	            "FC_Statistics"(ix_Reset := #iUDT_EquipmentControl.Command.ResetData,        // Reset statistics input
	                            ix_Activate := NOT #sx_safetyZoneOk,                                    // Activate statistics functions input
	                            ix_RTrigActivate := #sR_TRIG_NotHealthy.Q,                                   // Statistics active trigger
	                            iqUDT_Statistics := #iqUDT_Statistics.NotHealthy);                       // Statistics values output
	        END_IF;

	    END_REGION

	END_REGION



END_FUNCTION_BLOCK

FUNCTION_BLOCK "FB_UPSThreatParcel"
{ S7_Optimized_Access := 'TRUE' }
VERSION : 0.1
// ATTRIBUTES
// AUTO_NUMBER = True
// BLOCK_NUMBER = 63
// END_ATTRIBUTES
   VAR_INPUT
      ii_TrackingPosition { ExternalAccessible := 'False'; ExternalVisible := 'False'; ExternalWritable := 'False'} : Int;
      ix_ReleaseButton { ExternalAccessible := 'False'; ExternalVisible := 'False'; ExternalWritable := 'False'} : Bool;   // PSP release button
   END_VAR

   VAR_OUTPUT
      qx_StopConveyorDieBack { ExternalAccessible := 'False'; ExternalVisible := 'False'; ExternalWritable := 'False'} : Bool;   // Stop conveyor external die back
      qx_PreStopConveyorDieBack { ExternalAccessible := 'False'; ExternalVisible := 'False'; ExternalWritable := 'False'} : Bool;   // Pre stop conveyor external die back
      qx_ReleaseButtonIndication { ExternalAccessible := 'False'; ExternalVisible := 'False'; ExternalWritable := 'False'} : Bool;   // PSP release button indicator
      qx_Lamp { ExternalAccessible := 'False'; ExternalVisible := 'False'; ExternalWritable := 'False'} : Bool;   // Lamp indicator
      qx_HMIStatus { ExternalAccessible := 'False'; ExternalVisible := 'False'; ExternalWritable := 'False'} : Bool;
   END_VAR

   VAR_IN_OUT
      iqUDT_StopConveyorInterface : "UDT_ConveyorInterface";
      iqUDT_Handshake : "UDT_ConveyorHandshake";   // Conveyor handshake
      iqa_TrackingData : Array[*] of Int;   // Tracking array
   END_VAR

   VAR
      s_R_TRIG_ThreatParelFound {InstructionName := 'R_TRIG'; LibVersion := '1.0'; ExternalAccessible := 'False'; ExternalVisible := 'False'; ExternalWritable := 'False'; S7_SetPoint := 'False'} : R_TRIG;
      s_R_TRIG_Button {InstructionName := 'R_TRIG'; LibVersion := '1.0'; ExternalAccessible := 'False'; ExternalVisible := 'False'; ExternalWritable := 'False'; S7_SetPoint := 'False'} : R_TRIG;
      s_F_TRIG_Sensor {InstructionName := 'F_TRIG'; LibVersion := '1.0'; ExternalAccessible := 'False'; ExternalVisible := 'False'; ExternalWritable := 'False'; S7_SetPoint := 'False'} : F_TRIG;
      si_OldGIN { ExternalAccessible := 'False'; ExternalVisible := 'False'; ExternalWritable := 'False'} : Int;
      si_StopConveyorEmptyDistance { ExternalAccessible := 'False'; ExternalVisible := 'False'; ExternalWritable := 'False'} : Int;
      sx_ThreatParcelFound { ExternalAccessible := 'False'; ExternalVisible := 'False'; ExternalWritable := 'False'} : Bool;
      sx_SecondThreatParcelFound { ExternalAccessible := 'False'; ExternalVisible := 'False'; ExternalWritable := 'False'} : Bool;
      sx_StopConveyorEmpty { ExternalAccessible := 'False'; ExternalVisible := 'False'; ExternalWritable := 'False'} : Bool;
      sx_StopPreConveyor { ExternalAccessible := 'False'; ExternalVisible := 'False'; ExternalWritable := 'False'} : Bool;
   END_VAR


BEGIN
	(*
	----------------------------------------------------------------------------------------

	Version history:
	Date        | Version   | Author        | Remark
	----------------------------------------------------------------------------------------
	23/02/2021  | 0.1       | L.Klar        | first release MHS TIA 15.1
	22/02/2023  | 4.0       | F.Baten       | 4.0 Release TIA 17.5
	*)

	REGION 1 - Get new GIN

	    IF #iqa_TrackingData[#ii_TrackingPosition] > 0 AND
	        #iqa_TrackingData[#ii_TrackingPosition] <> #si_OldGIN
	    THEN

	        IF "DB_GIN".GIN[#iqa_TrackingData[#ii_TrackingPosition]].UPS.ThreatParcel THEN

	            IF #sx_ThreatParcelFound THEN
	                #sx_SecondThreatParcelFound := TRUE;
	            ELSE
	                #sx_ThreatParcelFound := TRUE;
	            END_IF;

	        END_IF;

	        #si_OldGIN := #iqa_TrackingData[#ii_TrackingPosition];
	    END_IF;

	    IF NOT #sx_ThreatParcelFound AND #sx_SecondThreatParcelFound THEN
	        #sx_ThreatParcelFound := TRUE;
	        #sx_SecondThreatParcelFound := FALSE;
	    END_IF;

	END_REGION

	REGION 2 - Release parcel

	    #s_R_TRIG_Button(CLK := #ix_ReleaseButton);

	    IF #s_R_TRIG_Button.Q THEN
	        #sx_ThreatParcelFound := FALSE;
	        #sx_StopConveyorEmpty := FALSE;
	        #sx_StopPreConveyor := FALSE;
	    END_IF;

	END_REGION



	REGION 2 - Threat parcel separtion

	    #s_R_TRIG_ThreatParelFound(CLK := #sx_ThreatParcelFound);
	    #s_F_TRIG_Sensor(CLK := #iqUDT_Handshake.TIP);

	    IF #s_R_TRIG_ThreatParelFound.Q THEN
	        #si_StopConveyorEmptyDistance := 300;
	    END_IF;

	    IF #si_StopConveyorEmptyDistance > 0 THEN
	        #si_StopConveyorEmptyDistance -= #iqUDT_StopConveyorInterface.Displacement;
	    END_IF;

	    IF #sx_ThreatParcelFound AND #si_StopConveyorEmptyDistance = 0 THEN
	        #sx_StopConveyorEmpty := TRUE;
	    END_IF;

	    IF #s_F_TRIG_Sensor.Q AND #sx_ThreatParcelFound AND #sx_StopConveyorEmpty THEN
	        #sx_StopPreConveyor := TRUE;
	        #sx_StopConveyorEmpty := FALSE;
	    END_IF;

	END_REGION

	REGION 3 - Outputs control

	    #qx_StopConveyorDieBack := #sx_ThreatParcelFound AND #sx_StopConveyorEmpty;
	    #qx_PreStopConveyorDieBack := ((#sx_ThreatParcelFound OR #sx_SecondThreatParcelFound) AND NOT #sx_StopConveyorEmpty) OR #sx_StopPreConveyor;

	    #qx_Lamp := #sx_ThreatParcelFound AND #sx_StopPreConveyor;
	    #qx_ReleaseButtonIndication := #sx_ThreatParcelFound AND #sx_StopPreConveyor;

	    #qx_HMIStatus := #sx_ThreatParcelFound AND #sx_StopPreConveyor;

	END_REGION
END_FUNCTION_BLOCK

FUNCTION_BLOCK "FB_UPS1stStageFlowControl"
{ S7_Optimized_Access := 'TRUE' }
VERSION : 0.1
// ATTRIBUTES
// AUTO_NUMBER = True
// BLOCK_NUMBER = 46
// END_ATTRIBUTES
   VAR_INPUT
      iUDT_configuration { ExternalAccessible := 'False'; ExternalVisible := 'False'; ExternalWritable := 'False'} : "UDT_UPS1stStageFlowControlConfiguration";   //   Configuration UDT
      idi_AdditionalRate { ExternalAccessible := 'False'; ExternalVisible := 'False'; ExternalWritable := 'False'} : DInt;   //   Additional rate from other measuring PLCs
      idi_ParcelCountInfeed1 { ExternalAccessible := 'False'; ExternalVisible := 'False'; ExternalWritable := 'False'} : DInt;   //   Counter of parcels from infeed
      ix_ActiveInfeed1 { ExternalAccessible := 'False'; ExternalVisible := 'False'; ExternalWritable := 'False'} : Bool;   //   Infeed is running / active
      idi_ParcelCountInfeed2 { ExternalAccessible := 'False'; ExternalVisible := 'False'; ExternalWritable := 'False'} : DInt;   //   Counter of parcels from infeed
      ix_ActiveInfeed2 { ExternalAccessible := 'False'; ExternalVisible := 'False'; ExternalWritable := 'False'} : Bool;   //   Infeed is running / active
      idi_ParcelCountInfeed3 { ExternalAccessible := 'False'; ExternalVisible := 'False'; ExternalWritable := 'False'} : DInt;   //   Counter of parcels from infeed
      ix_ActiveInfeed3 { ExternalAccessible := 'False'; ExternalVisible := 'False'; ExternalWritable := 'False'} : Bool;   //   Infeed is running / active
      idi_ParcelCountInfeed4 { ExternalAccessible := 'False'; ExternalVisible := 'False'; ExternalWritable := 'False'} : DInt;   //   Counter of parcels from infeed
      ix_ActiveInfeed4 { ExternalAccessible := 'False'; ExternalVisible := 'False'; ExternalWritable := 'False'} : Bool;   //   Infeed is running / active
      idi_ParcelCountInfeed5 { ExternalAccessible := 'False'; ExternalVisible := 'False'; ExternalWritable := 'False'} : DInt;   //   Counter of parcels from infeed
      ix_ActiveInfeed5 { ExternalAccessible := 'False'; ExternalVisible := 'False'; ExternalWritable := 'False'} : Bool;   //   Infeed is running / active
      idi_ParcelCountInfeed6 { ExternalAccessible := 'False'; ExternalVisible := 'False'; ExternalWritable := 'False'} : DInt;   //   Counter of parcels from infeed
      ix_ActiveInfeed6 { ExternalAccessible := 'False'; ExternalVisible := 'False'; ExternalWritable := 'False'} : Bool;   //   Infeed is running / active
      idi_ParcelCountInfeed7 { ExternalAccessible := 'False'; ExternalVisible := 'False'; ExternalWritable := 'False'} : DInt;   //   Counter of parcels from infeed
      ix_ActiveInfeed7 { ExternalAccessible := 'False'; ExternalVisible := 'False'; ExternalWritable := 'False'} : Bool;   //   Infeed is running / active
      idi_ParcelCountInfeed8 { ExternalAccessible := 'False'; ExternalVisible := 'False'; ExternalWritable := 'False'} : DInt;   //   Counter of parcels from infeed
      ix_ActiveInfeed8 { ExternalAccessible := 'False'; ExternalVisible := 'False'; ExternalWritable := 'False'} : Bool;   //   Infeed is running / active
      idi_ParcelCountInfeed9 { ExternalAccessible := 'False'; ExternalVisible := 'False'; ExternalWritable := 'False'} : DInt;   //   Counter of parcels from infeed
      ix_ActiveInfeed9 { ExternalAccessible := 'False'; ExternalVisible := 'False'; ExternalWritable := 'False'} : Bool;   //   Infeed is running / active
      idi_ParcelCountInfeed10 { ExternalAccessible := 'False'; ExternalVisible := 'False'; ExternalWritable := 'False'} : DInt;   //   Counter of parcels from infeed
      ix_ActiveInfeed10 { ExternalAccessible := 'False'; ExternalVisible := 'False'; ExternalWritable := 'False'} : Bool;   //   Infeed is running / active
   END_VAR

   VAR_OUTPUT
      qx_ConfigruationError { ExternalAccessible := 'False'; ExternalVisible := 'False'; ExternalWritable := 'False'} : Bool;   //   TRUE = Unexpected configuration
      qx_New15SecInterval { ExternalAccessible := 'False'; ExternalVisible := 'False'; ExternalWritable := 'False'} : Bool;   //   TRUE = Indicates a new 15 Sec interval to partner PLC
      qx_LimitFlowInfeed1 { ExternalAccessible := 'False'; ExternalVisible := 'False'; ExternalWritable := 'False'} : Bool;   //   TRUE = Stop infeed due flow control
      qdi_30secFlowInfeed1 { ExternalAccessible := 'False'; ExternalVisible := 'False'; ExternalWritable := 'False'} : DInt;   //   30 seconds pph rate
      qdi_1minFlowInfeed1 { ExternalAccessible := 'False'; ExternalVisible := 'False'; ExternalWritable := 'False'} : DInt;   //   1 minute pph rate
      qdi_3minFlowInfeed1 { ExternalAccessible := 'False'; ExternalVisible := 'False'; ExternalWritable := 'False'} : DInt;   //   3 minutes pph rate
      qdi_10minFlowInfeed1 { ExternalAccessible := 'False'; ExternalVisible := 'False'; ExternalWritable := 'False'} : DInt;   //   10 minutes pph rate
      qx_LimitFlowInfeed2 { ExternalAccessible := 'False'; ExternalVisible := 'False'; ExternalWritable := 'False'} : Bool;   //   TRUE = Stop infeed due flow control
      qdi_30secFlowInfeed2 { ExternalAccessible := 'False'; ExternalVisible := 'False'; ExternalWritable := 'False'} : DInt;   //   30 seconds pph rate
      qdi_1minFlowInfeed2 { ExternalAccessible := 'False'; ExternalVisible := 'False'; ExternalWritable := 'False'} : DInt;   //   1 minute pph rate
      qdi_3minFlowInfeed2 { ExternalAccessible := 'False'; ExternalVisible := 'False'; ExternalWritable := 'False'} : DInt;   //   3 minutes pph rate
      qdi_10minFlowInfeed2 { ExternalAccessible := 'False'; ExternalVisible := 'False'; ExternalWritable := 'False'} : DInt;   //   10 minutes pph rate
      qx_LimitFlowInfeed3 { ExternalAccessible := 'False'; ExternalVisible := 'False'; ExternalWritable := 'False'} : Bool;   //   TRUE = Stop infeed due flow control
      qdi_30secFlowInfeed3 { ExternalAccessible := 'False'; ExternalVisible := 'False'; ExternalWritable := 'False'} : DInt;   //   30 seconds pph rate
      qdi_1minFlowInfeed3 { ExternalAccessible := 'False'; ExternalVisible := 'False'; ExternalWritable := 'False'} : DInt;   //   1 minute pph rate
      qdi_3minFlowInfeed3 { ExternalAccessible := 'False'; ExternalVisible := 'False'; ExternalWritable := 'False'} : DInt;   //   3 minutes pph rate
      qdi_10minFlowInfeed3 { ExternalAccessible := 'False'; ExternalVisible := 'False'; ExternalWritable := 'False'} : DInt;   //   10 minutes pph rate
      qx_LimitFlowInfeed4 { ExternalAccessible := 'False'; ExternalVisible := 'False'; ExternalWritable := 'False'} : Bool;   //   TRUE = Stop infeed due flow control
      qdi_30secFlowInfeed4 { ExternalAccessible := 'False'; ExternalVisible := 'False'; ExternalWritable := 'False'} : DInt;   //   30 seconds pph rate
      qdi_1minFlowInfeed4 { ExternalAccessible := 'False'; ExternalVisible := 'False'; ExternalWritable := 'False'} : DInt;   //   1 minute pph rate
      qdi_3minFlowInfeed4 { ExternalAccessible := 'False'; ExternalVisible := 'False'; ExternalWritable := 'False'} : DInt;   //   3 minutes pph rate
      qdi_10minFlowInfeed4 { ExternalAccessible := 'False'; ExternalVisible := 'False'; ExternalWritable := 'False'} : DInt;   //   10 minutes pph rate
      qx_LimitFlowInfeed5 { ExternalAccessible := 'False'; ExternalVisible := 'False'; ExternalWritable := 'False'} : Bool;   //   TRUE = Stop infeed due flow control
      qdi_30secFlowInfeed5 { ExternalAccessible := 'False'; ExternalVisible := 'False'; ExternalWritable := 'False'} : DInt;   //   30 seconds pph rate
      qdi_1minFlowInfeed5 { ExternalAccessible := 'False'; ExternalVisible := 'False'; ExternalWritable := 'False'} : DInt;   //   1 minute pph rate
      qdi_3minFlowInfeed5 { ExternalAccessible := 'False'; ExternalVisible := 'False'; ExternalWritable := 'False'} : DInt;   //   3 minutes pph rate
      qdi_10minFlowInfeed5 { ExternalAccessible := 'False'; ExternalVisible := 'False'; ExternalWritable := 'False'} : DInt;   //   10 minutes pph rate
      qx_LimitFlowInfeed6 { ExternalAccessible := 'False'; ExternalVisible := 'False'; ExternalWritable := 'False'} : Bool;   //   TRUE = Stop infeed due flow control
      qdi_30secFlowInfeed6 { ExternalAccessible := 'False'; ExternalVisible := 'False'; ExternalWritable := 'False'} : DInt;   //   30 seconds pph rate
      qdi_1minFlowInfeed6 { ExternalAccessible := 'False'; ExternalVisible := 'False'; ExternalWritable := 'False'} : DInt;   //   1 minute pph rate
      qdi_3minFlowInfeed6 { ExternalAccessible := 'False'; ExternalVisible := 'False'; ExternalWritable := 'False'} : DInt;   //   3 minutes pph rate
      qdi_10minFlowInfeed6 { ExternalAccessible := 'False'; ExternalVisible := 'False'; ExternalWritable := 'False'} : DInt;   //   10 minutes pph rate
      qx_LimitFlowInfeed7 { ExternalAccessible := 'False'; ExternalVisible := 'False'; ExternalWritable := 'False'} : Bool;   //   TRUE = Stop infeed due flow control
      qdi_30secFlowInfeed7 { ExternalAccessible := 'False'; ExternalVisible := 'False'; ExternalWritable := 'False'} : DInt;   //   30 seconds pph rate
      qdi_1minFlowInfeed7 { ExternalAccessible := 'False'; ExternalVisible := 'False'; ExternalWritable := 'False'} : DInt;   //   1 minute pph rate
      qdi_3minFlowInfeed7 { ExternalAccessible := 'False'; ExternalVisible := 'False'; ExternalWritable := 'False'} : DInt;   //   3 minutes pph rate
      qdi_10minFlowInfeed7 { ExternalAccessible := 'False'; ExternalVisible := 'False'; ExternalWritable := 'False'} : DInt;   //   10 minutes pph rate
      qx_LimitFlowInfeed8 { ExternalAccessible := 'False'; ExternalVisible := 'False'; ExternalWritable := 'False'} : Bool;   //   TRUE = Stop infeed due flow control
      qdi_30secFlowInfeed8 { ExternalAccessible := 'False'; ExternalVisible := 'False'; ExternalWritable := 'False'} : DInt;   //   30 seconds pph rate
      qdi_1minFlowInfeed8 { ExternalAccessible := 'False'; ExternalVisible := 'False'; ExternalWritable := 'False'} : DInt;   //   1 minute pph rate
      qdi_3minFlowInfeed8 { ExternalAccessible := 'False'; ExternalVisible := 'False'; ExternalWritable := 'False'} : DInt;   //   3 minutes pph rate
      qdi_10minFlowInfeed8 { ExternalAccessible := 'False'; ExternalVisible := 'False'; ExternalWritable := 'False'} : DInt;   //   10 minutes pph rate
      qx_LimitFlowInfeed9 { ExternalAccessible := 'False'; ExternalVisible := 'False'; ExternalWritable := 'False'} : Bool;   //   TRUE = Stop infeed due flow control
      qdi_30secFlowInfeed9 { ExternalAccessible := 'False'; ExternalVisible := 'False'; ExternalWritable := 'False'} : DInt;   //   30 seconds pph rate
      qdi_1minFlowInfeed9 { ExternalAccessible := 'False'; ExternalVisible := 'False'; ExternalWritable := 'False'} : DInt;   //   1 minute pph rate
      qdi_3minFlowInfeed9 { ExternalAccessible := 'False'; ExternalVisible := 'False'; ExternalWritable := 'False'} : DInt;   //   3 minutes pph rate
      qdi_10minFlowInfeed9 { ExternalAccessible := 'False'; ExternalVisible := 'False'; ExternalWritable := 'False'} : DInt;   //   10 minutes pph rate
      qx_LimitFlowInfeed10 { ExternalAccessible := 'False'; ExternalVisible := 'False'; ExternalWritable := 'False'} : Bool;   //   TRUE = Stop infeed due flow control
      qdi_30secFlowInfeed10 { ExternalAccessible := 'False'; ExternalVisible := 'False'; ExternalWritable := 'False'} : DInt;   //   30 seconds pph rate
      qdi_1minFlowInfeed10 { ExternalAccessible := 'False'; ExternalVisible := 'False'; ExternalWritable := 'False'} : DInt;   //   1 minute pph rate
      qdi_3minFlowInfeed10 { ExternalAccessible := 'False'; ExternalVisible := 'False'; ExternalWritable := 'False'} : DInt;   //   3 minutes pph rate
      qdi_10minFlowInfeed10 { ExternalAccessible := 'False'; ExternalVisible := 'False'; ExternalWritable := 'False'} : DInt;   //   10 minutes pph rate
   END_VAR

   VAR_IN_OUT
      iqUDT_EquipmentControl : "UDT_EquipmentControl";
      iqUDT_FlowControlHMI : "UDT_UPSFlowControlHMI";
      iqa_InfeedArray : Array[1..10] of "UDT_UPSFlowRateCountingRegisters";   //   Array of line x
   END_VAR

   VAR
      sFB_Pulse_EndOf15sPeriod { ExternalAccessible := 'False'; ExternalVisible := 'False'; ExternalWritable := 'False'; S7_SetPoint := 'False'} : "FB_Pulse";   //   15 second pulse generator
      sa_infeed { ExternalAccessible := 'False'; ExternalVisible := 'False'; ExternalWritable := 'False'} : Array[1..10] of Struct   //   Data of infeed line
         diCounter { ExternalAccessible := 'False'; ExternalVisible := 'False'; ExternalWritable := 'False'} : DInt;   //   Counter of parcels from infeed
         diLastScanCounter { ExternalAccessible := 'False'; ExternalVisible := 'False'; ExternalWritable := 'False'} : DInt;   //   Last scan counter of parcels from infeed
         diFlowRate30sec { ExternalAccessible := 'False'; ExternalVisible := 'False'; ExternalWritable := 'False'} : DInt;   //   30sec pph rate
         diFlowRate1min { ExternalAccessible := 'False'; ExternalVisible := 'False'; ExternalWritable := 'False'} : DInt;   //   1 min pph rate
         diFlowRate3min { ExternalAccessible := 'False'; ExternalVisible := 'False'; ExternalWritable := 'False'} : DInt;   //   3 min pph rate
         diFlowRate10min { ExternalAccessible := 'False'; ExternalVisible := 'False'; ExternalWritable := 'False'} : DInt;   //   10 min pph rate
         iNumberOfNewParcels { ExternalAccessible := 'False'; ExternalVisible := 'False'; ExternalWritable := 'False'} : Int;   //   Number of new parcels during this scan
         Active { ExternalAccessible := 'False'; ExternalVisible := 'False'; ExternalWritable := 'False'} : Bool;   //   TRUE = infeed is active
         RequestStop { ExternalAccessible := 'False'; ExternalVisible := 'False'; ExternalWritable := 'False'} : Bool;   //   TRUE= Request flow control
         OneShotRequestStop { ExternalAccessible := 'False'; ExternalVisible := 'False'; ExternalWritable := 'False'} : Bool;   //   Rising edge request to stop
         DuringMinimumStopTime { ExternalAccessible := 'False'; ExternalVisible := 'False'; ExternalWritable := 'False'} : Bool;   //   Infeed is stopped and the minimum stop time is not elapsed
      END_STRUCT;
      sa_FirstToStop { ExternalAccessible := 'False'; ExternalVisible := 'False'; ExternalWritable := 'False'} : Array[1..10] of Int;   //   Number of infeed - sorted as per higher priotrity to stop
      sFB_MinStopTimeActive { ExternalAccessible := 'False'; ExternalVisible := 'False'; ExternalWritable := 'False'; S7_SetPoint := 'False'} : Array[1..10] of "FB_TimerOnOffDelay";   //   Minimum stop time active
      sdi_CumulativeFlowRate { ExternalAccessible := 'False'; ExternalVisible := 'False'; ExternalWritable := 'False'} : DInt;   //   Cumulative flow rate 1min pph at evaluation point
      sdi_AverageLength { ExternalAccessible := 'False'; ExternalVisible := 'False'; ExternalWritable := 'False'} : DInt;   //   Average length
      si_LastLowPriority { ExternalAccessible := 'False'; ExternalVisible := 'False'; ExternalWritable := 'False'} : Int;   //   Pointer to the last low priority infeed
      si_limit { ExternalAccessible := 'False'; ExternalVisible := 'False'; ExternalWritable := 'False'} : Int;   //   Number of infeeds in use - uper limit for array
      si_CurrentConsecutivesAboveSP { ExternalAccessible := 'False'; ExternalVisible := 'False'; ExternalWritable := 'False'} : Int;   //   Number of consecutive intervals  with flow above HMI set point
      si_CurrentConsecutivesBelowSP { ExternalAccessible := 'False'; ExternalVisible := 'False'; ExternalWritable := 'False'} : Int;   //   Number of consecutive intervals with flow below HMI set point
      sx_Disabled { ExternalAccessible := 'False'; ExternalVisible := 'False'; ExternalWritable := 'False'} : Bool;   //  Disabled from user
      sx_StopRequested { ExternalAccessible := 'False'; ExternalVisible := 'False'; ExternalWritable := 'False'} : Bool;   //   Any infeed requested to stop
      sx_swapLowPriority { ExternalAccessible := 'False'; ExternalVisible := 'False'; ExternalWritable := 'False'} : Bool;   //   Used to indicate swap of position in the priority sorting
      sx_swapHighPriority { ExternalAccessible := 'False'; ExternalVisible := 'False'; ExternalWritable := 'False'} : Bool;   //   Used to indicate swap of position in the priority sorting
   END_VAR

   VAR_TEMP
      tr_quotient : Real;   //   Quotient of division
      tr_fraction : Real;   //   Return of fraction
      ti_buffer : Int;   //   Auxiliary buffer
      ti_LC_i : Int;   //   Loop counter
      ti_LC_k : Int;   //   Loop counter
      ti_Index : Int;   //   temporaty index
      ti_HighPriorityLowLimit : Int;   //   pointer to high priority low limit
      tx_End15sPeriod : Bool;   //   End of 15 seconds flow period
      tx_invalidLimit : Bool;   //   Invalid number of diverts
      tx_invalidOffset : Bool;   //   Invalid offset in a divert
   END_VAR

   VAR CONSTANT
      cdi_InchesAverageLength : DInt := DINT#20;   //   Average length in inches
      cdi_mmAverageLength : DInt := DINT#508;   //   Average length in mm
   END_VAR


BEGIN
	(*
	----------------------------------------------------------------------------------------

	Version history:
	Date        | Version   | Author        | Remark
	----------------------------------------------------------------------------------------
	09/04/2020  | 3.0       | S.Theocharis  | First release. UPS Appendix B V2.0 20161010
	22/04/2020  | 3.1       | S.Theocharis  | Changed to handle product length
	24/04/2020  | 3.2       | S.Theocharis  | Convert INTs to DINTs.
	                                        | Add validation check for negative offset
	24/04/2020  | 3.3       | S.Theocharis  | Bug fix of the index used in 1min flow calculation
	29/04/2020  | 3.4       | K.Pokorski    | Change prefix to qdi so as to match variable types
	28/01/2021  | 3.5       | S.Theocharis  | Update HMI interface. Add disable command and disabled status
	10/04/2021  | 3.6       | S.Theocharis  | Add input additional flow to evaluated flow. For inbound area
	21/02/2023  | 4.0       | F.Baten       | 4.0 Release TIA 17.5
	13/03/2024  | 4.1       | S. Nieświec   | 4.1 Release TIA 18
	*)

	REGION 1 - Normalization and data move

	    REGION 1.1 - Normalization

	        IF #iUDT_configuration.LegthBasedFlowControl THEN

	            IF #iUDT_configuration.IsLengthImperial THEN
	                #sdi_AverageLength := #cdi_InchesAverageLength;  // infeed count in inches
	            ELSE
	                #sdi_AverageLength := #cdi_mmAverageLength;       // infeed count in mm
	            END_IF;
	        ELSE
	            #sdi_AverageLength := L#1;                            // infeed count in parcels
	        END_IF;

	    END_REGION

	    REGION 1.2 - Move Input data to static
	        //Move counters
	        #sa_infeed[1].diCounter := #idi_ParcelCountInfeed1;
	        #sa_infeed[2].diCounter := #idi_ParcelCountInfeed2;
	        #sa_infeed[3].diCounter := #idi_ParcelCountInfeed3;
	        #sa_infeed[4].diCounter := #idi_ParcelCountInfeed4;
	        #sa_infeed[5].diCounter := #idi_ParcelCountInfeed5;
	        #sa_infeed[6].diCounter := #idi_ParcelCountInfeed6;
	        #sa_infeed[7].diCounter := #idi_ParcelCountInfeed7;
	        #sa_infeed[8].diCounter := #idi_ParcelCountInfeed8;
	        #sa_infeed[9].diCounter := #idi_ParcelCountInfeed9;
	        #sa_infeed[10].diCounter := #idi_ParcelCountInfeed10;

	        //Move infeed active bit
	        #sa_infeed[1].Active := #ix_ActiveInfeed1;
	        #sa_infeed[2].Active := #ix_ActiveInfeed2;
	        #sa_infeed[3].Active := #ix_ActiveInfeed3;
	        #sa_infeed[4].Active := #ix_ActiveInfeed4;
	        #sa_infeed[5].Active := #ix_ActiveInfeed5;
	        #sa_infeed[6].Active := #ix_ActiveInfeed6;
	        #sa_infeed[7].Active := #ix_ActiveInfeed7;
	        #sa_infeed[8].Active := #ix_ActiveInfeed8;
	        #sa_infeed[9].Active := #ix_ActiveInfeed9;

	        //map number of infeeds in use at the static memory
	        #si_limit := #iUDT_configuration.NumberOfInfeedsInUse;

	    END_REGION

	END_REGION

	REGION 2 - Validate configuration
	    //We validate configuration in every scan...
	    //..validation on first scan is also possible

	    //Check number of used diverts
	    #tx_invalidLimit := #si_limit <= 1
	    OR #si_limit > 10;

	    //Check divert offset configuration
	    //the offset cannot be above 56 because it will lead outside of the array size when we calculate the cummulative flow rate
	    IF NOT #tx_invalidLimit THEN
	        FOR #ti_LC_i := 1 TO #si_limit BY 1 DO
	            IF
	                #iUDT_configuration.Infeed[#ti_LC_i].RegisterOffset > 56 OR #iUDT_configuration.Infeed[#ti_LC_i].RegisterOffset < 0
	            THEN
	                #tx_invalidOffset := TRUE;
	            END_IF;
	        END_FOR;
	    END_IF;

	    // Error handling
	    IF #tx_invalidLimit OR #tx_invalidOffset OR #iUDT_configuration.IntervalsNumberOfEvaluationPeriod = 0 THEN
	        //On error: Set error output..
	        #qx_ConfigruationError := TRUE;

	        //..reset flow control outputs..
	        #qx_LimitFlowInfeed1 := FALSE;
	        #qx_LimitFlowInfeed2 := FALSE;
	        #qx_LimitFlowInfeed3 := FALSE;
	        #qx_LimitFlowInfeed4 := FALSE;
	        #qx_LimitFlowInfeed5 := FALSE;
	        #qx_LimitFlowInfeed6 := FALSE;
	        #qx_LimitFlowInfeed7 := FALSE;
	        #qx_LimitFlowInfeed8 := FALSE;
	        #qx_LimitFlowInfeed9 := FALSE;
	        #qx_LimitFlowInfeed10 := FALSE;

	        //..and exit block
	        RETURN;
	    ELSE
	        #qx_ConfigruationError := FALSE;
	    END_IF;

	END_REGION

	REGION 3 - End of 15s flow period

	    // Calculate 15 seconds period
	    #sFB_Pulse_EndOf15sPeriod(iudi_PulseTime := 15000,
	                              qx_Pulse => #tx_End15sPeriod);

	END_REGION

	REGION 4 - Add number of parcels in the register
	    //Each Region is used for different configurations

	    REGION 4.1 - When input counts are incrementing

	        IF #iUDT_configuration.IncrementingCounts THEN

	            FOR #ti_LC_i := 1 TO #si_limit BY 1 DO

	                //calculate new parcels per infeed
	                IF #sa_infeed[#ti_LC_i].diCounter >= #sa_infeed[#ti_LC_i].diLastScanCounter THEN
	                    //Parcels are incremented normaly
	                    #sa_infeed[#ti_LC_i].iNumberOfNewParcels := DINT_TO_INT(#sa_infeed[#ti_LC_i].diCounter - #sa_infeed[#ti_LC_i].diLastScanCounter);

	                ELSE
	                    //Exception handling of parcel counter was reset in the partner PLC. Therefore for this scan we don't subtrack the ones of the previous scan
	                    #sa_infeed[#ti_LC_i].iNumberOfNewParcels := DINT_TO_INT(#sa_infeed[#ti_LC_i].diCounter);
	                END_IF;

	                //Move current counter at the static variable of the last scan
	                #sa_infeed[#ti_LC_i].diLastScanCounter := #sa_infeed[#ti_LC_i].diCounter;

	                //add new parcels in the 1st register
	                #iqa_InfeedArray[#ti_LC_i].iCR[1] += (#sa_infeed[#ti_LC_i].iNumberOfNewParcels);

	            END_FOR;
	        END_IF;

	    END_REGION

	    REGION 4.2 - When input counts are updated every 15 sec interval
	        //That logic here needs to be tested. There is a risk of loosing some parcels beacuse of the delay between the pLC to PLC communication.

	        IF NOT #iUDT_configuration.IncrementingCounts AND #tx_End15sPeriod THEN

	            FOR #ti_LC_i := 1 TO #si_limit BY 1 DO

	                #iqa_InfeedArray[#ti_LC_i].iCR[1] := DINT_TO_INT(#sa_infeed[#ti_LC_i].diCounter);

	            END_FOR;

	        END_IF;
	    END_REGION

	END_REGION

	REGION 5 - Flow rate calculation
	    // The 15 second period has passed
	    IF (#tx_End15sPeriod) THEN

	        // loop the used infeeds
	        FOR #ti_LC_i := 1 TO #si_limit BY 1 DO

	            // Initialize static flow buffer
	            #sa_infeed[#ti_LC_i].diFlowRate30sec := L#0;
	            #sa_infeed[#ti_LC_i].diFlowRate1min := L#0;
	            #sa_infeed[#ti_LC_i].diFlowRate3min := L#0;
	            #sa_infeed[#ti_LC_i].diFlowRate10min := L#0;

	            // Loop through 40 Counting Registers per infeed
	            FOR #ti_LC_k := 1 TO 40 DO

	                // 30 sec flow handling
	                IF #ti_LC_k <= 2 THEN
	                    #sa_infeed[#ti_LC_i].diFlowRate30sec += INT_TO_DINT(#iqa_InfeedArray[#ti_LC_i].iCR[#ti_LC_k]);

	                    // Conversion to full hour
	                    IF #ti_LC_k = 2
	                    THEN
	                        #sa_infeed[#ti_LC_i].diFlowRate30sec *= L#120;

	                        //Normalise
	                        #sa_infeed[#ti_LC_i].diFlowRate30sec /= #sdi_AverageLength;


	                    END_IF;
	                END_IF;

	                // 1 minute flow handling
	                IF #ti_LC_k <= 4 THEN
	                    #sa_infeed[#ti_LC_i].diFlowRate1min += INT_TO_DINT(#iqa_InfeedArray[#ti_LC_i].iCR[#ti_LC_k]);

	                    // Conversion to full hour
	                    IF #ti_LC_k = 4 THEN
	                        #sa_infeed[#ti_LC_i].diFlowRate1min *= L#60;
	                        //Normalise
	                        #sa_infeed[#ti_LC_i].diFlowRate1min /= #sdi_AverageLength;
	                    END_IF;
	                END_IF;

	                // 3 minutes flow handling
	                IF #ti_LC_k <= 12 THEN
	                    #sa_infeed[#ti_LC_i].diFlowRate3min += INT_TO_DINT(#iqa_InfeedArray[#ti_LC_i].iCR[#ti_LC_k]);

	                    // Conversion to full hour
	                    IF #ti_LC_k = 12 THEN
	                        #sa_infeed[#ti_LC_i].diFlowRate3min *= L#20;
	                        //Normalise
	                        #sa_infeed[#ti_LC_i].diFlowRate3min /= #sdi_AverageLength;
	                    END_IF;
	                END_IF;

	                // 10 minutes flow handling
	                #sa_infeed[#ti_LC_i].diFlowRate10min += INT_TO_DINT(#iqa_InfeedArray[#ti_LC_i].iCR[#ti_LC_k]);

	                // Conversion to full hour
	                IF #ti_LC_k = 40
	                THEN
	                    #sa_infeed[#ti_LC_i].diFlowRate10min *= L#6;
	                    //Normalise
	                    #sa_infeed[#ti_LC_i].diFlowRate10min /= #sdi_AverageLength;
	                END_IF;

	            END_FOR;

	        END_FOR;

	    END_IF;

	END_REGION

	REGION 6 - Cumulative flow at evaluation point

	    IF (#tx_End15sPeriod) THEN

	        //initialise static variable
	        #sdi_CumulativeFlowRate := L#0;

	        FOR #ti_LC_i := 1 TO #si_limit BY 1 DO

	            FOR #ti_LC_k := 1 TO 4 BY 1 DO

	                #sdi_CumulativeFlowRate += INT_TO_DINT(#iqa_InfeedArray[#ti_LC_i].iCR[#ti_LC_k + #iUDT_configuration.Infeed[#ti_LC_i].RegisterOffset]);

	            END_FOR;

	        END_FOR;

	        // Conversion to full hour
	        #sdi_CumulativeFlowRate *= L#60;

	        //Normalise
	        #sdi_CumulativeFlowRate /= #sdi_AverageLength;

	        //add additional rate calculated in other PLCs ( e.g. recirculation OTE RATE!)
	        #sdi_CumulativeFlowRate := #sdi_CumulativeFlowRate + #idi_AdditionalRate;



	    END_IF;

	END_REGION

	REGION 7 - Shift arrays when 15s flow period ends

	    // 15 seconds period elapsed
	    IF (#tx_End15sPeriod) THEN

	        FOR #ti_LC_i := 1 TO #si_limit BY 1 DO

	            // Shifted counting register by one element down
	            MOVE_BLK(IN := #iqa_InfeedArray[#ti_LC_i].iCR[1],
	                     COUNT := 59,
	                     OUT => #iqa_InfeedArray[#ti_LC_i].iCR[2]);

	            // Reset first registter
	            #iqa_InfeedArray[#ti_LC_i].iCR[1] := 0;

	        END_FOR;
	    END_IF;

	END_REGION

	REGION 8 - Compare Current Value with Set Point

	    IF (#tx_End15sPeriod) THEN

	        IF #sdi_CumulativeFlowRate >= INT_TO_DINT(#iqUDT_FlowControlHMI.Setpoint) THEN

	            #si_CurrentConsecutivesAboveSP += 1;  //increment consecutives above set point
	            #si_CurrentConsecutivesBelowSP := 0;  //reset consecutives below set point
	        ELSE

	            #si_CurrentConsecutivesAboveSP := 0;  //reset consecutives above set point
	            #si_CurrentConsecutivesBelowSP += 1;  //increment consecutives below set point

	            //limit consecutives below set point to threshold value. Protection against INT overflow
	            IF #si_CurrentConsecutivesBelowSP >= #iUDT_configuration.ThresholdConsecutivesBelowSP THEN

	                #si_CurrentConsecutivesBelowSP := #iUDT_configuration.ThresholdConsecutivesBelowSP;

	            END_IF;

	        END_IF;

	    END_IF;

	END_REGION

	REGION 9 - Evaluation - Apply flow control
	    //The evaluation period is specified by UPS at 1min or 4 intervals of 15 seconds

	    IF (#tx_End15sPeriod) AND #si_CurrentConsecutivesAboveSP > 0 THEN

	        //divide  current consecutives above SP with the number of intervals for evaluation ,,
	        #tr_quotient := INT_TO_REAL(#si_CurrentConsecutivesAboveSP) / INT_TO_REAL(#iUDT_configuration.IntervalsNumberOfEvaluationPeriod);

	        //call fraction to check the number of decimal places of the quotient
	        #tr_fraction := FRAC(#tr_quotient);

	        //If there are no decimal places then the current consecutive above set point is multiple
	        //of the evaluation period. Therefore the evaluation of the flow control should take place.
	        IF #tr_fraction = 0.0 THEN

	            REGION 9.1 - Sort infeeds from 1st to stop to last to stop
	                //Sort as per priorities. From low priority to high
	                //The high priority infeeds will be last in the sort regardless their flow

	                //initialize index
	                #ti_Index := 1;

	                //Sort from top the low priority infeeds
	                FOR #ti_LC_i := 1 TO #si_limit BY 1 DO

	                    IF #iUDT_configuration.Infeed[#ti_LC_i].IsHighPriority = FALSE THEN
	                        #sa_FirstToStop[#ti_Index] := #ti_LC_i;
	                        #ti_Index += 1;
	                    END_IF;

	                END_FOR;

	                //Pointer to last low priority infeed
	                #si_LastLowPriority := #ti_Index - 1;

	                //Sort the high priority infeeds if there are any
	                IF #si_LastLowPriority < #si_limit THEN
	                    FOR #ti_LC_i := 1 TO #si_limit BY 1 DO

	                        IF #iUDT_configuration.Infeed[#ti_LC_i].IsHighPriority = TRUE THEN
	                            #sa_FirstToStop[#ti_Index] := #ti_LC_i;
	                            #ti_Index += 1;
	                        END_IF;

	                    END_FOR;
	                END_IF;

	                //Sort based on the flow. Low priority infeeds
	                IF #si_LastLowPriority > 0 THEN

	                    REPEAT
	                        #sx_swapLowPriority := FALSE;

	                        FOR #ti_LC_i := #si_LastLowPriority TO 2 BY -1 DO
	                            IF #sa_infeed[#sa_FirstToStop[#ti_LC_i - 1]].diFlowRate1min < #sa_infeed[#sa_FirstToStop[#ti_LC_i]].diFlowRate1min THEN

	                                #ti_buffer := #sa_FirstToStop[#ti_LC_i];
	                                #sa_FirstToStop[#ti_LC_i] := #sa_FirstToStop[#ti_LC_i - 1];
	                                #sa_FirstToStop[#ti_LC_i - 1] := #ti_buffer;
	                                #sx_swapLowPriority := TRUE;

	                            END_IF;
	                        END_FOR;
	                    UNTIL NOT #sx_swapLowPriority
	                    END_REPEAT;
	                END_IF;


	                //Sort based on the flow. High priority infeeds
	                IF #si_LastLowPriority < #si_limit THEN
	                    #ti_HighPriorityLowLimit := (#si_LastLowPriority + 1);
	                    REPEAT
	                        #sx_swapHighPriority := FALSE;

	                        FOR #ti_LC_i := #si_limit TO #ti_HighPriorityLowLimit BY -1 DO

	                            IF (#sa_infeed[#sa_FirstToStop[#ti_LC_i - 1]].diFlowRate1min < #sa_infeed[#sa_FirstToStop[#ti_LC_i]].diFlowRate1min)
	                                AND #iUDT_configuration.Infeed[#sa_FirstToStop[#ti_LC_i - 1]].IsHighPriority
	                            THEN

	                                #ti_buffer := #sa_FirstToStop[#ti_LC_i];
	                                #sa_FirstToStop[#ti_LC_i] := #sa_FirstToStop[#ti_LC_i - 1];
	                                #sa_FirstToStop[#ti_LC_i - 1] := #ti_buffer;
	                                #sx_swapHighPriority := TRUE;

	                            END_IF;
	                        END_FOR;
	                    UNTIL NOT #sx_swapHighPriority
	                    END_REPEAT;
	                END_IF;

	            END_REGION

	            REGION 9.2 - Request stop to limit flow

	                FOR #ti_LC_i := 1 TO #si_limit BY 1 DO

	                    IF
	                        #sa_infeed[#sa_FirstToStop[#ti_LC_i]].Active                                      //infeed running / activated ..
	                        AND NOT #sa_infeed[#sa_FirstToStop[#ti_LC_i]].RequestStop                            // .. and not already stopped...
	                        AND NOT #sa_infeed[#sa_FirstToStop[#ti_LC_i]].DuringMinimumStopTime                  // .. and not during minimum time to stop
	                        AND NOT #iUDT_configuration.Infeed[#sa_FirstToStop[#ti_LC_i]].IsNotAllowedToStop    // and is allowed to stop.

	                    THEN
	                        #sa_infeed[#sa_FirstToStop[#ti_LC_i]].RequestStop := TRUE;
	                        #sa_infeed[#sa_FirstToStop[#ti_LC_i]].OneShotRequestStop := TRUE;
	                        EXIT;                                                                                   //exit loop to stop one infeed every evaluation interval
	                    END_IF;

	                END_FOR;

	            END_REGION

	        END_IF;

	    END_IF;

	END_REGION

	REGION 10 - Evaluation - Remove flow control

	    IF (#tx_End15sPeriod) AND #si_CurrentConsecutivesBelowSP >= #iUDT_configuration.ThresholdConsecutivesBelowSP THEN

	        FOR #ti_LC_i := 1 TO #si_limit BY 1 DO
	            #sa_infeed[#ti_LC_i].RequestStop := FALSE;
	        END_FOR;

	    END_IF;

	END_REGION

	REGION 11  - Set minimum time of stopped time

	    FOR #ti_LC_i := 1 TO #si_limit BY 1 DO

	        //Set minimum time to stop
	        #sFB_MinStopTimeActive[#ti_LC_i](iudi_OnDelayTime := 0,
	                                         iudi_OffDelayTime := #iUDT_configuration.Infeed[#ti_LC_i].MinimumTimeToStop,
	                                         ix_SignalToDelay := #sa_infeed[#ti_LC_i].OneShotRequestStop,
	                                         ix_Enable := TRUE,
	                                         qx_DelayedSignal => #sa_infeed[#ti_LC_i].DuringMinimumStopTime);

	        //reset one shot request to stop
	        #sa_infeed[#ti_LC_i].OneShotRequestStop := FALSE;

	    END_FOR;

	END_REGION

	REGION 12 - HMI Enable / Disable

	    //Command to disable frlow control from HMI
	    #sx_Disabled := #iqUDT_FlowControlHMI.CommandToDisable;

	END_REGION

	REGION 12 - Ouput the request stop

	    #qx_LimitFlowInfeed1 := (#sa_infeed[1].RequestStop OR #sa_infeed[1].DuringMinimumStopTime) AND NOT #sx_Disabled;
	    #qx_LimitFlowInfeed2 := (#sa_infeed[2].RequestStop OR #sa_infeed[2].DuringMinimumStopTime) AND NOT #sx_Disabled;
	    #qx_LimitFlowInfeed3 := (#sa_infeed[3].RequestStop OR #sa_infeed[3].DuringMinimumStopTime) AND NOT #sx_Disabled;
	    #qx_LimitFlowInfeed4 := (#sa_infeed[4].RequestStop OR #sa_infeed[4].DuringMinimumStopTime) AND NOT #sx_Disabled;
	    #qx_LimitFlowInfeed5 := (#sa_infeed[5].RequestStop OR #sa_infeed[5].DuringMinimumStopTime) AND NOT #sx_Disabled;
	    #qx_LimitFlowInfeed6 := (#sa_infeed[6].RequestStop OR #sa_infeed[6].DuringMinimumStopTime) AND NOT #sx_Disabled;
	    #qx_LimitFlowInfeed7 := (#sa_infeed[7].RequestStop OR #sa_infeed[7].DuringMinimumStopTime) AND NOT #sx_Disabled;
	    #qx_LimitFlowInfeed8 := (#sa_infeed[8].RequestStop OR #sa_infeed[8].DuringMinimumStopTime) AND NOT #sx_Disabled;
	    #qx_LimitFlowInfeed9 := (#sa_infeed[9].RequestStop OR #sa_infeed[9].DuringMinimumStopTime) AND NOT #sx_Disabled;
	    #qx_LimitFlowInfeed10 := (#sa_infeed[10].RequestStop OR #sa_infeed[10].DuringMinimumStopTime) AND NOT #sx_Disabled;

	END_REGION

	REGION 13 - Output flow rates

	    //Disabled status to HMI
	    #iqUDT_FlowControlHMI.DisabledStatus := #sx_Disabled;

	    ///Output 15 Sec interval one shot
	    #qx_New15SecInterval := #tx_End15sPeriod;

	    //Cumulative
	    #iqUDT_FlowControlHMI.CalculatedFlow := DINT_TO_INT(#sdi_CumulativeFlowRate);

	    //Infeed 1
	    #qdi_30secFlowInfeed1 := (#sa_infeed[1].diFlowRate30sec);
	    #qdi_1minFlowInfeed1 := (#sa_infeed[1].diFlowRate1min);
	    #qdi_3minFlowInfeed1 := (#sa_infeed[1].diFlowRate3min);
	    #qdi_10minFlowInfeed1 := (#sa_infeed[1].diFlowRate10min);

	    //Infeed 2
	    #qdi_30secFlowInfeed2 := (#sa_infeed[2].diFlowRate30sec);
	    #qdi_1minFlowInfeed2 := (#sa_infeed[2].diFlowRate1min);
	    #qdi_3minFlowInfeed2 := (#sa_infeed[2].diFlowRate3min);
	    #qdi_10minFlowInfeed2 := (#sa_infeed[2].diFlowRate10min);

	    //Infeed 3
	    #qdi_30secFlowInfeed3 := (#sa_infeed[3].diFlowRate30sec);
	    #qdi_1minFlowInfeed3 := (#sa_infeed[3].diFlowRate1min);
	    #qdi_3minFlowInfeed3 := (#sa_infeed[3].diFlowRate3min);
	    #qdi_10minFlowInfeed3 := (#sa_infeed[3].diFlowRate10min);

	    //Infeed 4
	    #qdi_30secFlowInfeed4 := (#sa_infeed[4].diFlowRate30sec);
	    #qdi_1minFlowInfeed4 := (#sa_infeed[4].diFlowRate1min);
	    #qdi_3minFlowInfeed4 := (#sa_infeed[4].diFlowRate3min);
	    #qdi_10minFlowInfeed4 := (#sa_infeed[4].diFlowRate10min);

	    //Infeed 5
	    #qdi_30secFlowInfeed5 := (#sa_infeed[5].diFlowRate30sec);
	    #qdi_1minFlowInfeed5 := (#sa_infeed[5].diFlowRate1min);
	    #qdi_3minFlowInfeed5 := (#sa_infeed[5].diFlowRate3min);
	    #qdi_10minFlowInfeed5 := (#sa_infeed[5].diFlowRate10min);

	    //Infeed 6
	    #qdi_30secFlowInfeed6 := (#sa_infeed[6].diFlowRate30sec);
	    #qdi_1minFlowInfeed6 := (#sa_infeed[6].diFlowRate1min);
	    #qdi_3minFlowInfeed6 := (#sa_infeed[6].diFlowRate3min);
	    #qdi_10minFlowInfeed6 := (#sa_infeed[6].diFlowRate10min);

	    //Infeed 7
	    #qdi_30secFlowInfeed7 := (#sa_infeed[7].diFlowRate30sec);
	    #qdi_1minFlowInfeed7 := (#sa_infeed[7].diFlowRate1min);
	    #qdi_3minFlowInfeed7 := (#sa_infeed[7].diFlowRate3min);
	    #qdi_10minFlowInfeed7 := (#sa_infeed[7].diFlowRate10min);

	    //Infeed 8
	    #qdi_30secFlowInfeed8 := (#sa_infeed[8].diFlowRate30sec);
	    #qdi_1minFlowInfeed8 := (#sa_infeed[8].diFlowRate1min);
	    #qdi_3minFlowInfeed8 := (#sa_infeed[8].diFlowRate3min);
	    #qdi_10minFlowInfeed8 := (#sa_infeed[8].diFlowRate10min);

	    //Infeed 9
	    #qdi_30secFlowInfeed9 := (#sa_infeed[9].diFlowRate30sec);
	    #qdi_1minFlowInfeed9 := (#sa_infeed[9].diFlowRate1min);
	    #qdi_3minFlowInfeed9 := (#sa_infeed[9].diFlowRate3min);
	    #qdi_10minFlowInfeed9 := (#sa_infeed[9].diFlowRate10min);

	    //Infeed 10
	    #qdi_30secFlowInfeed10 := (#sa_infeed[10].diFlowRate30sec);
	    #qdi_1minFlowInfeed10 := (#sa_infeed[10].diFlowRate1min);
	    #qdi_3minFlowInfeed10 := (#sa_infeed[10].diFlowRate3min);
	    #qdi_10minFlowInfeed10 := (#sa_infeed[10].diFlowRate10min);

	END_REGION

END_FUNCTION_BLOCK

